// TIA Portal V18 export
// export: Created 2026-06-16T05:09:48.2267058Z, ExportSetting WithDefaults, DisplayName Totally Integrated Automation Portal, DisplayVersion V18 Update 5, DisplayName TIA Portal Openness, DisplayVersion V18 Update 5, DisplayName TIA Portal Version Control Interface, DisplayVersion V18, DisplayName SINAMICS Startdrive Advanced, DisplayVersion V18 SP2 Update 1, DisplayName SINAMICS Startdrive G110M, G120, G120C, G120D, G120P, G115D, DisplayVersion V18 SP2 Update 1, DisplayName SINAMICS Startdrive G130, G150, S120, S150, SINAMICS MV, S210, G220, S200, DisplayVersion V18 SP2 Update 1, DisplayName STEP 7 Professional, DisplayVersion V18 Update 5, DisplayName STEP 7 Safety, DisplayVersion V18, DisplayName WinCC Advanced / Unified PC, DisplayVersion V18 Update 5
FUNCTION "TEMPLATE--v1.1--02_EM Push Button" : Void   // FC5, F_LAD
TITLE = Mirror PB
{ S7_Optimized_Access := 'TRUE' }
VERSION : 0.1
// v1.0 First emission
// 1.1 Aligned Syntax to signal_types.csv of the py_builder
// stored: AutoNumber true, IsIECCheckEnabled false, UDAEnableTagReadback false
BEGIN

REGION Network 1: !!NetworkComment$$
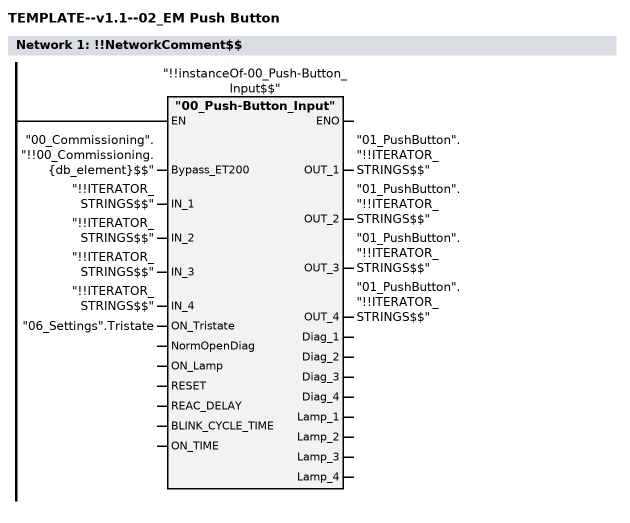
   RUNG wire#powerrail
      "!!instanceOf-00_Push-Button_Input$$"(Bypass_ET200 := "00_Commissioning"."!!00_Commissioning.{db_element}$$", IN_1 := "!!ITERATOR_STRINGS$$", IN_2 := "!!ITERATOR_STRINGS$$", IN_3 := "!!ITERATOR_STRINGS$$", IN_4 := "!!ITERATOR_STRINGS$$", ON_Tristate := "06_Settings".Tristate, NormOpenDiag :=, ON_Lamp :=, RESET :=, REAC_DELAY :=, BLINK_CYCLE_TIME :=, ON_TIME :=, OUT_1 => "01_PushButton"."!!ITERATOR_STRINGS$$", OUT_2 => "01_PushButton"."!!ITERATOR_STRINGS$$", OUT_3 => "01_PushButton"."!!ITERATOR_STRINGS$$", OUT_4 => "01_PushButton"."!!ITERATOR_STRINGS$$", Diag_1 =>, Diag_2 =>, Diag_3 =>, Diag_4 =>, Lamp_1 =>, Lamp_2 =>, Lamp_3 =>, Lamp_4 =>)
   END_RUNG
   // the same network as SCL:
   "!!instanceOf-00_Push-Button_Input$$"(Bypass_ET200 := "00_Commissioning"."!!00_Commissioning.{db_element}$$",   // "00_Push-Button_Input"
                           IN_1 := "!!ITERATOR_STRINGS$$",
                           IN_2 := "!!ITERATOR_STRINGS$$",
                           IN_3 := "!!ITERATOR_STRINGS$$",
                           IN_4 := "!!ITERATOR_STRINGS$$",
                           ON_Tristate := "06_Settings".Tristate,
                           OUT_1 => "01_PushButton"."!!ITERATOR_STRINGS$$",
                           OUT_2 => "01_PushButton"."!!ITERATOR_STRINGS$$",
                           OUT_3 => "01_PushButton"."!!ITERATOR_STRINGS$$",
                           OUT_4 => "01_PushButton"."!!ITERATOR_STRINGS$$");
END_REGION
END_FUNCTION
